% RSLogix 500 project Job 22 - Leo Kniffen.RSS, saved by version 10.00.00.00 %
PROJECT "ML04B"    % processor: Bul.1763 MicroLogix 1100 Series B %

PROGRAM FILES
  LAD 2   7 rungs

DATA FILES
  O0 OUTPUT  4 elements
  I1 INPUT  6 elements
  S2 STATUS  66 elements
  B3 BINARY  1 elements
  T4 TIMER  1 elements
  C5 COUNTER  1 elements
  R6 CONTROL  1 elements
  N7 INTEGER  1 elements
  F8 FLOAT  1 elements

LADDER 2
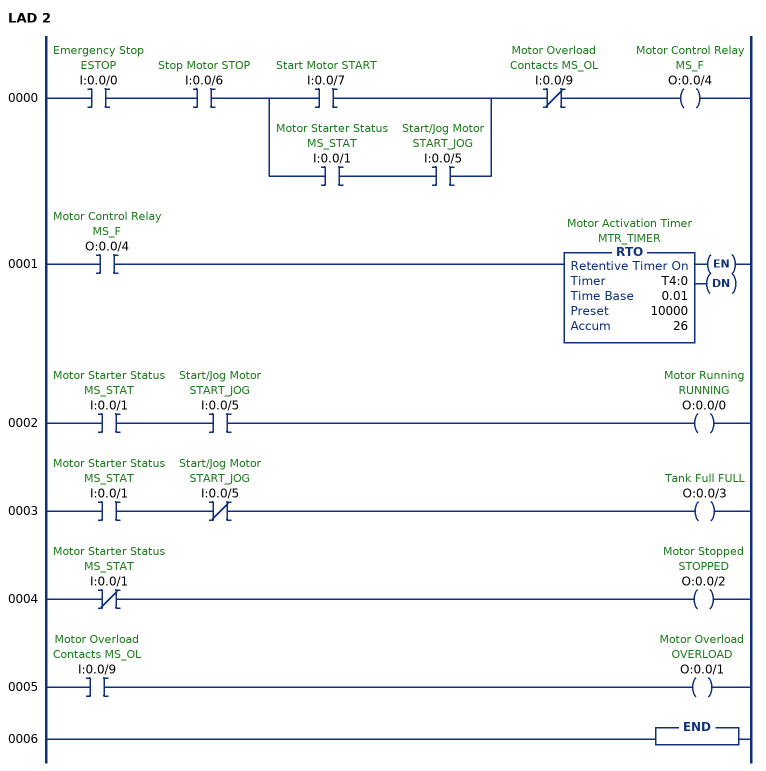
% Rung: 0 %
SOR XIC I:0.0/0 XIC I:0.0/6 BST XIC I:0.0/7 NXB XIC I:0.0/1 XIC I:0.0/5 BND XIO I:0.0/9 OTE O:0.0/4 EOR
%   I:0.0/0  ESTOP  "Emergency Stop" %
%   I:0.0/6  STOP  "Stop Motor" %
%   I:0.0/7  START  "Start Motor" %
%   I:0.0/1  MS_STAT  "Motor Starter Status" %
%   I:0.0/5  START_JOG  "Start/Jog Motor" %
%   I:0.0/9  MS_OL  "Motor Overload Contacts" %
%   O:0.0/4  MS_F  "Motor Control Relay" %
% Rung: 1 %
SOR XIC O:0.0/4 RTO T4:0 0.01 10000 26 EOR
%   O:0.0/4  MS_F  "Motor Control Relay" %
%   T4:0  MTR_TIMER  "Motor Activation Timer" %
% Rung: 2 %
SOR XIC I:0.0/1 XIC I:0.0/5 OTE O:0.0/0 EOR
%   I:0.0/1  MS_STAT  "Motor Starter Status" %
%   I:0.0/5  START_JOG  "Start/Jog Motor" %
%   O:0.0/0  RUNNING  "Motor Running" %
% Rung: 3 %
SOR XIC I:0.0/1 XIO I:0.0/5 OTE O:0.0/3 EOR
%   I:0.0/1  MS_STAT  "Motor Starter Status" %
%   I:0.0/5  START_JOG  "Start/Jog Motor" %
%   O:0.0/3  FULL  "Tank Full" %
% Rung: 4 %
SOR XIO I:0.0/1 OTE O:0.0/2 EOR
%   I:0.0/1  MS_STAT  "Motor Starter Status" %
%   O:0.0/2  STOPPED  "Motor Stopped" %
% Rung: 5 %
SOR XIC I:0.0/9 OTE O:0.0/1 EOR
%   I:0.0/9  MS_OL  "Motor Overload Contacts" %
%   O:0.0/1  OVERLOAD  "Motor Overload" %
% Rung: 6 %
SOR END EOR

OTHER DOCUMENTED ADDRESSES
  B3:0/0  VLV_AUTO  "Valve Control Bit"
  B3:0/1  VLV_ON  "Valve Cotrol Bit"
  B3:0/2  JOG_BIT  "Motor Control/Jog"
  B3:0/3  REV_SAVED  "Saved reverse bit"
  I:0.0/2  DIR_STAT  "Motor Direction Status"
  I:0.0/3  MODE_AUTO  "Mode, On/Off/Auto"
  I:0.0/4  MODE_ON  "Mode, On/Off/Auto"
  I:0.0/8  JOG  "Jog Motor"
  O:0.0/5  CR2  "Direction Control Relay"
  T4  
  T4:0.ACC/0  FLASH  "Flashing Bit"
  T4:0/DN  TIMER_D  "Timer Done"
  T4:0/EN  TIMER_E  "Timer enable"
  T4:0/TT  TIMER_ON  "Accumulation Active"

COMMENTS NOT ATTACHED TO A CURRENT RUNG
  B3:0/0: Job 18: Deadband Tank Level Control
    Leo Kniffen

DATA TABLE (non-zero values as saved)
DATA B3
% B3:0 % 0X0002
DATA T4
% .PRE .ACC %
% T4:0 % 10000 26
